// SIMATIC STEP 7 (V5.x) project Two Motors One Button
// CPU: CPU 314C-2 DP
// station: Hardware
// station: SIMATIC 300(1)
// station: P_ADR_BUS
// program: S7 Program(1)

SYMBOL_TABLE
"Button"	I 0.0	BOOL
"Motor1"	Q 0.0	BOOL
"Motor2"	Q 0.1	BOOL
END_SYMBOL_TABLE

ORGANIZATION_BLOCK OB 1
TITLE = "Two Motors and One Button"
VERSION : 0.1
VAR_TEMP
  OB1_EV_CLASS : BYTE ;	//Bits 0-3 = 1 (Coming event), Bits 4-7 = 1 (Event class 1)
  OB1_SCAN_1 : BYTE ;	//1 (Cold restart scan 1 of OB 1), 3 (Scan 2-n of OB 1)
  OB1_PRIORITY : BYTE ;	//Priority of OB Execution
  OB1_OB_NUMBR : BYTE ;	//1 (Organization block 1, OB1)
  OB1_RESERVED_1 : BYTE ;	//Reserved for system
  OB1_RESERVED_2 : BYTE ;	//Reserved for system
  OB1_PREV_CYCLE : INT ;	//Cycle time of previous OB1 scan (milliseconds)
  OB1_MIN_CYCLE : INT ;	//Minimum cycle time of OB1 (milliseconds)
  OB1_MAX_CYCLE : INT ;	//Maximum cycle time of OB1 (milliseconds)
  OB1_DATE_TIME : DATE_AND_TIME ;	//Date and time OB1 started
END_VAR
BEGIN
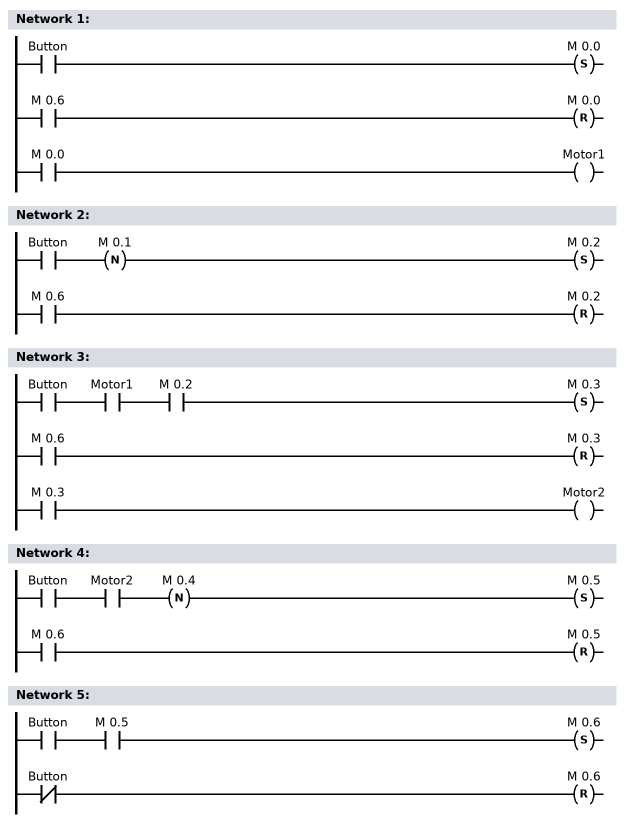
NETWORK
TITLE =
      A     "Button";
      S     M 0.0;
      A     M 0.6;
      R     M 0.0;
      A     M 0.0;
      =     "Motor1";
NETWORK
TITLE =
      A     "Button";
      FN    M 0.1;
      S     M 0.2;
      A     M 0.6;
      R     M 0.2;
      NOP   0;
NETWORK
TITLE =
      A     "Button";
      A     "Motor1";
      A     M 0.2;
      S     M 0.3;
      A     M 0.6;
      R     M 0.3;
      A     M 0.3;
      =     "Motor2";
NETWORK
TITLE =
      A     "Button";
      A     "Motor2";
      FN    M 0.4;
      S     M 0.5;
      A     M 0.6;
      R     M 0.5;
      NOP   0;
NETWORK
TITLE =
      A     "Button";
      A     M 0.5;
      S     M 0.6;
      AN    "Button";
      R     M 0.6;
      NOP   0;
END_ORGANIZATION_BLOCK
